Staubli VAL3: test.dtx

mdesc mNomSpeed
tool tTool = {z=110, fatherId=flange[0], ioLink=valve1}
jointRx jAproachPiece = {j1=-5.03067209967487, j2=43.3081121684082, j3=54.1351709463615, j4=4.70507356684578, j5=79.1734286699559, j6=-42.7327028817804}
jointRx jHome
pointRx pGetObject = {x=535.528546033673, y=9.14839041231438, z=-274.924251333, rx=-0.71666123620136, ry=179.698141439783, rz=-36.8198549749438, fatherId=world[0]}
